FUNCTION URL_DECODE : T_MaxString
VAR_INPUT
	IN : T_MaxString;
END_VAR
VAR
	pos : INT;
	seq : STRING(3);
	new : STRING(1);
END_VAR


(*
version 1.2		10. may. 2010
programmer 	hugo
tested by		hugo

URL_DECODE checks a string if it contains non reserved characters represented by a % followed with the two digit hex code and converts them to their ascii code.
the non reserved characters are : [A..Z], [a..z], [0..9], -_.~
for example the character sequence '%23' will be converted to '#'.

*)

URL_DECODE := IN;
pos := FIND(URL_DECODE,'%');
WHILE pos > 0 DO
	seq := MID(URL_DECODE,2,pos + 1);
	new := CHR_TO_STRING(DWORD_TO_BYTE(HEX_TO_DWORD(seq)));
	URL_DECODE := REPLACE(URL_DECODE, new, 3, pos);
	pos := FIND(URL_DECODE,'%');
END_WHILE;


(* revision history
hm	27. apr. 2008	rev 1.0
	original version

hm	17. dec. 2008	rev 1.1
	changes name of function chr to chr_to_string

ks	10. mai. 2008	rev 1.2
	stringlength 250
*)

END_FUNCTION

(* stored: Version 1.1.0.1, ProductVersion 3.1.4024.9
   POU URL_DECODE: Id {deb925fa-fe5e-4743-9e8a-872581a3ed96}, SpecialFunc None *)
